(* Schneider Machine Expert - Basic project Exercise-3 - Multiple Switch Connection for LEDs, file version 2.9.0.0 *)
(* ProjectInformations: Name=New project *)

HARDWARE
  Cpu 0: TM221C24R
  EthernetConfiguration: NetworkName=M221, IpAllocationMode=FixedAddress, IpAddress=0.0.0.0, SubnetMask=0.0.0.0
  SerialLineConfiguration: Baud=Baud19200, Parity=ParityEven, DataBits=DataBits8, StopBits=StopBits1, PhysicalMedium=PhysicalMediumRs485, SlaveId=1, Addressing=SlaveAddressing
  MastTask: UsePeriodScanMode=false, PeriodScan=100
  FastTask: Period=255
  CpuBehavior: StartingMode=StartAsPreviousState, AutoSaveRamOnEeprom=true, WatchdogPeriod=250

SYMBOLS  (address, symbol, comment, settings)
  %I0.0     SWITCH_1
  %I0.1     SWITCH_2
  %I0.2     SWITCH_3
  %Q0.0     LED_1
  %Q0.1     LED_2
  %Q0.2     LED_3

POU New POU
  (* SectionNumber=1 *)

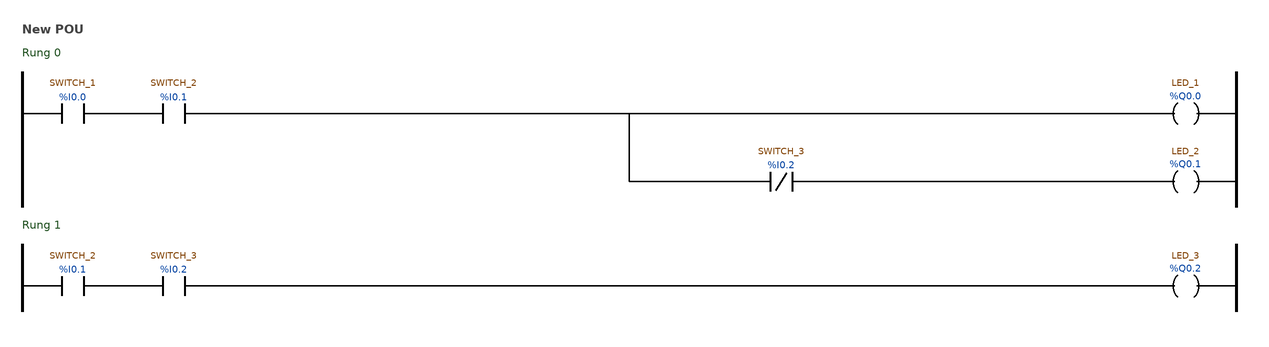

// Rung 0
  LD %I0.0                (* SWITCH_1 *)
  AND %I0.1               (* SWITCH_2 *)
  MPS
  ST %Q0.0                (* LED_1 *)
  MPP
  ANDN %I0.2              (* SWITCH_3 *)
  ST %Q0.1                (* LED_2 *)
  // as ST:
  //   LED_1 := SWITCH_1 AND SWITCH_2;
  //   LED_2 := SWITCH_1 AND SWITCH_2 AND NOT SWITCH_3;

// Rung 1
  LD %I0.1                (* SWITCH_2 *)
  AND %I0.2               (* SWITCH_3 *)
  ST %Q0.2                (* LED_3 *)
  // as ST:
  //   LED_3 := SWITCH_2 AND SWITCH_3;
